(* CoDeSys 2.3.9.47 project: wtp_sfc_6_1_2016.pro *)
(* Libraries: TcSystem.lib 21.1.15 10:22:54, TcBase.lib 14.5.09 12:14:08, TcUtilities.lib 6.1.15 16:45:04, TcBABasic.lib 22.7.15 15:46:14, STANDARD.LIB 5.6.98 12:03:02 *)

(* Task configuration *)
TASK Standard (PRIORITY := 0, INTERVAL := T#500ms);
	MAIN
END_TASK

(* POU MAIN, ST *)
PROGRAM MAIN
VAR
(*EQUALISATION TRANSFER*)

	InletEqPumpOp1 :  INLET_EQ_PUMP;

	LSL101A: BOOL;
	LSS101A: BOOL;
	LSH101A: BOOL;
	LSD101A: BOOL;
	LSHH105A: BOOL;
	LSH103A: BOOL;
	LSS103A: BOOL;

	InletEqPumpOp2 :  INLET_EQ_PUMP;

	LSL101B: BOOL;
	LSS101B: BOOL;
	LSH101B: BOOL;
	LSD101B: BOOL;
	LSHH105B: BOOL;
	LSH103B: BOOL;
	LSS103B: BOOL;


	InletMixerOp1 : INLET_MIXER;
	LSL100A : BOOL;
	LSHL100A : BOOL;

	InletMixerOp2 : INLET_MIXER;
	LSL100B : BOOL;
	LSHL100B : BOOL;


(*SBR TRANSFER*)
	SBRTrans_OP1_InletSBRTrans : INLET_EQ_PUMP;
	SBRTrans_OP2_InletSBRTrans : INLET_EQ_PUMP;

	test : DEVICES_DOUBLE_DUTY;
	WaterPressureSensor: REAL;

(*Reuse Water Syatem*)
	Reuse_Water_System : REUSE_WATER_SYS;

(*Screen House*)
	ScreenOperation1 : SCREENING_OPERATION;


END_VAR
(*EQUALISATION TRANSFER*)
InletEqPumpOp1(
	sigEQFloatSensorLO:= LSL101A,
	sigEQFLoatSensorOP:= LSS101A,
	sigEQFloatSensorHi:= LSH101A,
	sigEQFLoatSensorDry:= LSD101A,
	sigStreamLineOverFLow:=LSHH105A ,
	sigSBRFloatSensorHi:= LSH103A,
	sigSBRFloatSensorOP:=LSS103A );

InletEqPumpOp2(
	sigEQFloatSensorLO:= LSL101B,
	sigEQFLoatSensorOP:= LSS101B,
	sigEQFloatSensorHi:= LSH101B,
	sigEQFLoatSensorDry:= LSD101B,
	sigStreamLineOverFLow:=LSHH105B ,
	sigSBRFloatSensorHi:= LSH103B,
	sigSBRFloatSensorOP:=LSS103B );

InletMixerOp1(sigMixerFloatSensorLO:=LSL100A , sigMixerFloatSensorHI:=LSHL100A );

InletMixerOp2(sigMixerFloatSensorLO:=LSL100B , sigMixerFloatSensorHI:=LSHL100B );



(*Reuse Water Syatem*)
	Reuse_Water_System();



(*Screen House*)
ScreenOperation1();
END_PROGRAM

(* POU INLET_EQ_PUMP, SFC *)
FUNCTION_BLOCK  INLET_EQ_PUMP
VAR

	Reset : BOOL;
	CriticalAlarm_FloatSensorHi : BOOL;
	CriticalAlarm_FloatSensorDRY : BOOL;
	Warning_FloatSensorDry : BOOL;


	Pump : DEVICES_DUTY_STANDBY;

	Act_Reset : BOOL;
	Act_Start : BOOL;
	Act_Stop : BOOL;

	FB_Contacts_1: FB_Contacts;
	FB_Contacts_2:FB_Contacts;
	FB_Contacts_3:FB_Contacts;
	FB_Contacts_4:FB_Contacts;
	FB_Contacts_5:FB_Contacts;
	FB_Contacts_6:FB_Contacts;
	FB_Contacts_7:FB_Contacts;


	EQFloatSensorLO : BOOL;
	EQFLoatSensorOP : BOOL;
	EQFloatSensorHi : BOOL;
	EQFLoatSensorDry : BOOL;
	StreamLineOverFLow : BOOL;
	SBRFloatSensorHi : BOOL;
	SBRFloatSensorOP : BOOL;
END_VAR
VAR_IN_OUT
	sigEQFloatSensorLO : BOOL;
	sigEQFLoatSensorOP : BOOL;
	sigEQFloatSensorHi : BOOL;
	sigEQFLoatSensorDry : BOOL;
	sigStreamLineOverFLow : BOOL;
	sigSBRFloatSensorHi : BOOL;
	sigSBRFloatSensorOP : BOOL;
END_VAR
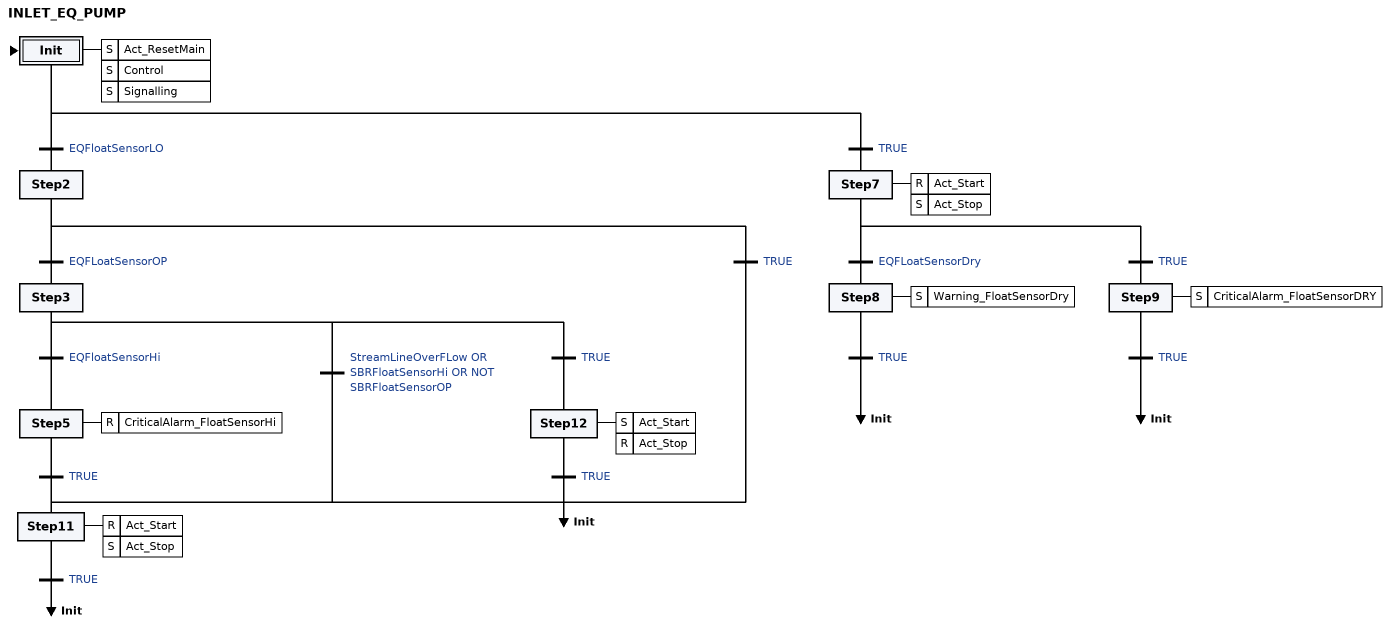
INITIAL_STEP Init:
	Act_ResetMain(S);
	Control(S);
	Signalling(S);
END_STEP
TRANSITION FROM Init TO Step2 := EQFloatSensorLO;
END_TRANSITION
TRANSITION FROM Init TO Step7 := TRUE;
END_TRANSITION
STEP Step2:
END_STEP
TRANSITION FROM Step2 TO Step3 := EQFLoatSensorOP;
END_TRANSITION
TRANSITION FROM Step2 TO Step11 := TRUE;
END_TRANSITION
STEP Step3:
END_STEP
TRANSITION FROM Step3 TO Step5 := EQFloatSensorHi;
END_TRANSITION
TRANSITION FROM Step3 TO Step11 := StreamLineOverFLow OR SBRFloatSensorHi OR NOT SBRFloatSensorOP;
END_TRANSITION
TRANSITION FROM Step3 TO Step12 := TRUE;
END_TRANSITION
STEP Step5:
	CriticalAlarm_FloatSensorHi(R);
END_STEP
TRANSITION FROM Step5 TO Step11 := TRUE;
END_TRANSITION
STEP Step11:
	Act_Start(R);
	Act_Stop(S);
END_STEP
TRANSITION FROM Step11 TO Init := TRUE;
END_TRANSITION
STEP Step12:
	Act_Start(S);
	Act_Stop(R);
END_STEP
TRANSITION FROM Step12 TO Init := TRUE;
END_TRANSITION
STEP Step7:
	Act_Start(R);
	Act_Stop(S);
END_STEP
TRANSITION FROM Step7 TO Step8 := EQFLoatSensorDry;
END_TRANSITION
TRANSITION FROM Step7 TO Step9 := TRUE;
END_TRANSITION
STEP Step8:
	Warning_FloatSensorDry(S);
END_STEP
TRANSITION FROM Step8 TO Init := TRUE;
END_TRANSITION
STEP Step9:
	CriticalAlarm_FloatSensorDRY(S);
END_STEP
TRANSITION FROM Step9 TO Init := TRUE;
END_TRANSITION
END_FUNCTION_BLOCK
ACTION Act_ResetMain:
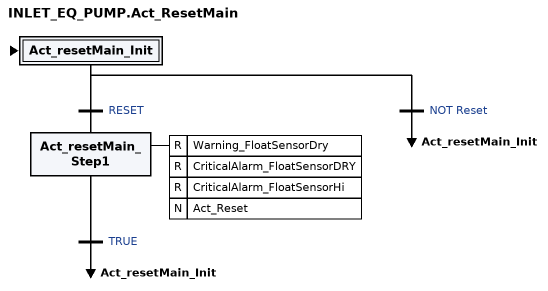
INITIAL_STEP Act_resetMain_Init:
END_STEP
TRANSITION FROM Act_resetMain_Init TO Act_resetMain_Step1 := RESET;
END_TRANSITION
TRANSITION FROM Act_resetMain_Init TO Act_resetMain_Init := NOT Reset;
END_TRANSITION
STEP Act_resetMain_Step1:
	Warning_FloatSensorDry(R);
	CriticalAlarm_FloatSensorDRY(R);
	CriticalAlarm_FloatSensorHi(R);
	Act_Reset(N);
END_STEP
TRANSITION FROM Act_resetMain_Step1 TO Act_resetMain_Init := TRUE;
END_TRANSITION
END_ACTION
ACTION Control:
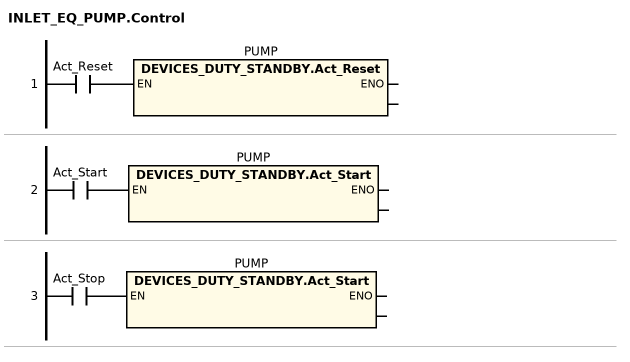
_LD_ (* Ladder Diagram *)
NETWORK 1
	[Act_Reset]
		EN --- PUMP:DEVICES_DUTY_STANDBY.Act_Reset()
NETWORK 2
	[Act_Start]
		EN --- PUMP:DEVICES_DUTY_STANDBY.Act_Start()
NETWORK 3
	[Act_Stop]
		EN --- PUMP:DEVICES_DUTY_STANDBY.Act_Start()
_END_LD_
(* the same logic as Structured Text *)
(* Network 1 *)
IF Act_Reset THEN
	PUMP();
END_IF;
(* Network 2 *)
IF Act_Start THEN
	PUMP();
END_IF;
(* Network 3 *)
IF Act_Stop THEN
	PUMP();
END_IF;
END_ACTION
ACTION Signalling:
FB_Contacts_1(IN:=sigEQFloatSensorLO ,Q=> EQFloatSensorLO);
FB_Contacts_2(IN:=sigEQFLoatSensorOP ,Q=> EQFLoatSensorOP);
FB_Contacts_3(IN:=sigEQFloatSensorHi ,Q=> EQFloatSensorHi);
FB_Contacts_4(IN:=sigEQFLoatSensorDry ,Q=> EQFLoatSensorDry);
FB_Contacts_5(IN:=sigStreamLineOverFLow ,Q=> StreamLineOverFLow);
FB_Contacts_6(IN:=sigSBRFloatSensorHi ,Q=> SBRFloatSensorHi);
FB_Contacts_7(IN:=sigSBRFloatSensorOP ,Q=> SBRFloatSensorOP);
END_ACTION

(* POU DEVICES_DUTY_STANDBY, SFC *)
FUNCTION_BLOCK DEVICES_DUTY_STANDBY
VAR


	Duty_RemoteMode AT%I*: BOOL;
	Duty_CommandStart AT%I*: BOOL;
	Duty_Overload AT%I*: BOOL;
	Duty_Incomplete AT%I*: BOOL;
	Duty_StartStatus AT%I*: BOOL;


	Done_StartStandby: BOOL;
	Done_Start: BOOL;
	Done_Stop: BOOL;


	Standby_CommandStart AT%I*: BOOL;
	Standby_RemoteMode AT%I*: BOOL;
	Standby_Overload AT%I*: BOOL;
	Standby_Incomplete AT%I*: BOOL;
	Standby_StartStatus AT%I*: BOOL;


	Warning_DutyFailed: BOOL;
	Warning_StandbyFailed: BOOL;
	CriticalAlarm_StandbyCannotStop : BOOL;
	CriticalAlarm_DutyCannotStop : BOOL;
	CriticalAlarm_DutyStandbyFailedToStart: BOOL;

END_VAR
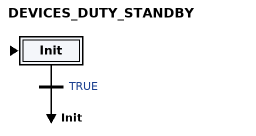
INITIAL_STEP Init:
END_STEP
TRANSITION FROM Init TO Init := TRUE;
END_TRANSITION
END_FUNCTION_BLOCK
ACTION Act_Reset:
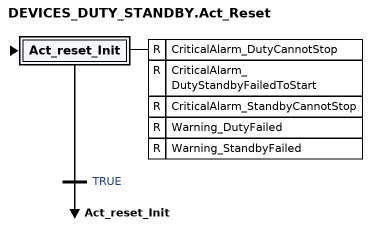
INITIAL_STEP Act_reset_Init:
	CriticalAlarm_DutyCannotStop(R);
	CriticalAlarm_DutyStandbyFailedToStart(R);
	CriticalAlarm_StandbyCannotStop(R);
	Warning_DutyFailed(R);
	Warning_StandbyFailed(R);
END_STEP
TRANSITION FROM Act_reset_Init TO Act_reset_Init := TRUE;
END_TRANSITION
END_ACTION
ACTION Act_Start:
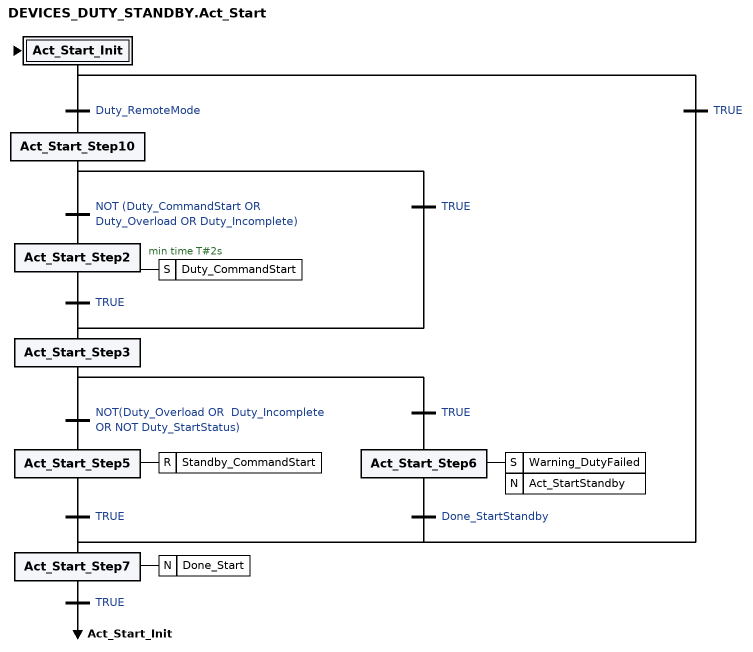
INITIAL_STEP Act_Start_Init:
END_STEP
TRANSITION FROM Act_Start_Init TO Act_Start_Step10 := Duty_RemoteMode;
END_TRANSITION
TRANSITION FROM Act_Start_Init TO Act_Start_Step7 := TRUE;
END_TRANSITION
STEP Act_Start_Step10:
END_STEP
TRANSITION FROM Act_Start_Step10 TO Act_Start_Step2 := NOT (Duty_CommandStart OR Duty_Overload OR Duty_Incomplete);
END_TRANSITION
TRANSITION FROM Act_Start_Step10 TO Act_Start_Step3 := TRUE;
END_TRANSITION
STEP Act_Start_Step2: (* min time T#2s *)
	Duty_CommandStart(S);
END_STEP
TRANSITION FROM Act_Start_Step2 TO Act_Start_Step3 := TRUE;
END_TRANSITION
STEP Act_Start_Step3:
END_STEP
TRANSITION FROM Act_Start_Step3 TO Act_Start_Step5 := NOT(Duty_Overload OR  Duty_Incomplete OR NOT Duty_StartStatus);
END_TRANSITION
TRANSITION FROM Act_Start_Step3 TO Act_Start_Step6 := TRUE;
END_TRANSITION
STEP Act_Start_Step5:
	Standby_CommandStart(R);
END_STEP
TRANSITION FROM Act_Start_Step5 TO Act_Start_Step7 := TRUE;
END_TRANSITION
STEP Act_Start_Step6:
	Warning_DutyFailed(S);
	Act_StartStandby(N);
END_STEP
TRANSITION FROM Act_Start_Step6 TO Act_Start_Step7 := Done_StartStandby;
END_TRANSITION
STEP Act_Start_Step7:
	Done_Start(N);
END_STEP
TRANSITION FROM Act_Start_Step7 TO Act_Start_Init := TRUE;
END_TRANSITION
END_ACTION
ACTION Act_StartStandby:
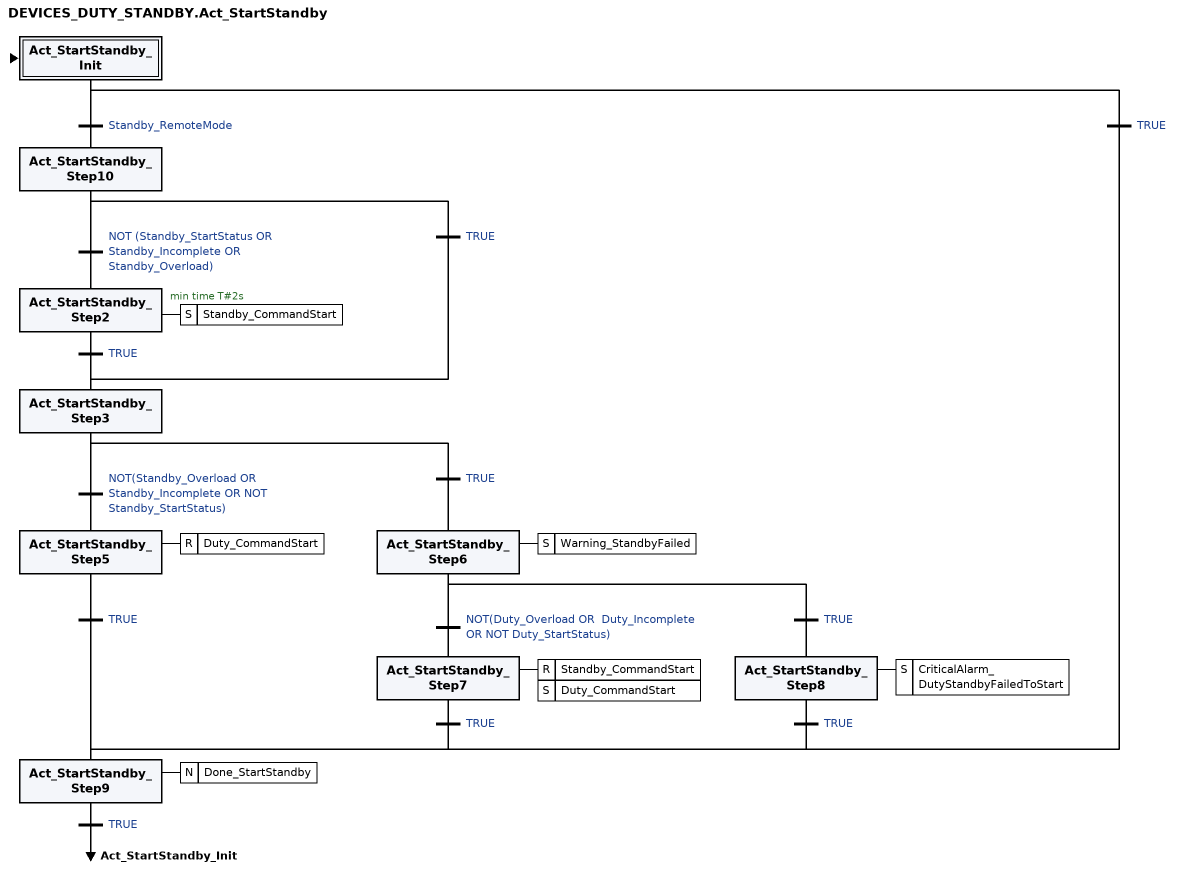
INITIAL_STEP Act_StartStandby_Init:
END_STEP
TRANSITION FROM Act_StartStandby_Init TO Act_StartStandby_Step10 := Standby_RemoteMode;
END_TRANSITION
TRANSITION FROM Act_StartStandby_Init TO Act_StartStandby_Step9 := TRUE;
END_TRANSITION
STEP Act_StartStandby_Step10:
END_STEP
TRANSITION FROM Act_StartStandby_Step10 TO Act_StartStandby_Step2 := NOT (Standby_StartStatus OR Standby_Incomplete OR Standby_Overload);
END_TRANSITION
TRANSITION FROM Act_StartStandby_Step10 TO Act_StartStandby_Step3 := TRUE;
END_TRANSITION
STEP Act_StartStandby_Step2: (* min time T#2s *)
	Standby_CommandStart(S);
END_STEP
TRANSITION FROM Act_StartStandby_Step2 TO Act_StartStandby_Step3 := TRUE;
END_TRANSITION
STEP Act_StartStandby_Step3:
END_STEP
TRANSITION FROM Act_StartStandby_Step3 TO Act_StartStandby_Step5 := NOT(Standby_Overload OR  Standby_Incomplete OR NOT Standby_StartStatus);
END_TRANSITION
TRANSITION FROM Act_StartStandby_Step3 TO Act_StartStandby_Step6 := TRUE;
END_TRANSITION
STEP Act_StartStandby_Step5:
	Duty_CommandStart(R);
END_STEP
TRANSITION FROM Act_StartStandby_Step5 TO Act_StartStandby_Step9 := TRUE;
END_TRANSITION
STEP Act_StartStandby_Step6:
	Warning_StandbyFailed(S);
END_STEP
TRANSITION FROM Act_StartStandby_Step6 TO Act_StartStandby_Step7 := NOT(Duty_Overload OR  Duty_Incomplete OR NOT Duty_StartStatus);
END_TRANSITION
TRANSITION FROM Act_StartStandby_Step6 TO Act_StartStandby_Step8 := TRUE;
END_TRANSITION
STEP Act_StartStandby_Step7:
	Standby_CommandStart(R);
	Duty_CommandStart(S);
END_STEP
TRANSITION FROM Act_StartStandby_Step7 TO Act_StartStandby_Step9 := TRUE;
END_TRANSITION
STEP Act_StartStandby_Step8:
	CriticalAlarm_DutyStandbyFailedToStart (S);
END_STEP
TRANSITION FROM Act_StartStandby_Step8 TO Act_StartStandby_Step9 := TRUE;
END_TRANSITION
STEP Act_StartStandby_Step9:
	Done_StartStandby(N);
END_STEP
TRANSITION FROM Act_StartStandby_Step9 TO Act_StartStandby_Init := TRUE;
END_TRANSITION
END_ACTION
ACTION Act_Stop:
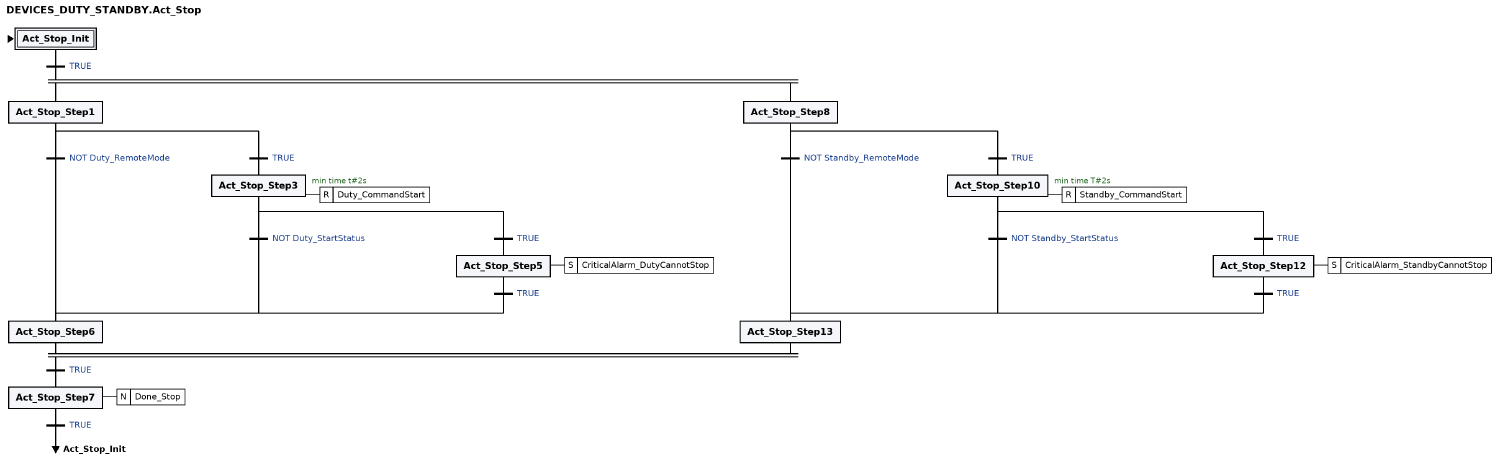
INITIAL_STEP Act_Stop_Init:
END_STEP
TRANSITION FROM Act_Stop_Init TO (Act_Stop_Step1, Act_Stop_Step8) := TRUE;
END_TRANSITION
STEP Act_Stop_Step1:
END_STEP
TRANSITION FROM Act_Stop_Step1 TO Act_Stop_Step6 := NOT Duty_RemoteMode;
END_TRANSITION
TRANSITION FROM Act_Stop_Step1 TO Act_Stop_Step3 := TRUE;
END_TRANSITION
STEP Act_Stop_Step3: (* min time t#2s *)
	Duty_CommandStart(R);
END_STEP
TRANSITION FROM Act_Stop_Step3 TO Act_Stop_Step6 := NOT Duty_StartStatus;
END_TRANSITION
TRANSITION FROM Act_Stop_Step3 TO Act_Stop_Step5 := TRUE;
END_TRANSITION
STEP Act_Stop_Step5:
	CriticalAlarm_DutyCannotStop(S);
END_STEP
TRANSITION FROM Act_Stop_Step5 TO Act_Stop_Step6 := TRUE;
END_TRANSITION
STEP Act_Stop_Step6:
END_STEP
STEP Act_Stop_Step8:
END_STEP
TRANSITION FROM Act_Stop_Step8 TO Act_Stop_Step13 := NOT Standby_RemoteMode;
END_TRANSITION
TRANSITION FROM Act_Stop_Step8 TO Act_Stop_Step10 := TRUE;
END_TRANSITION
STEP Act_Stop_Step10: (* min time T#2s *)
	Standby_CommandStart(R);
END_STEP
TRANSITION FROM Act_Stop_Step10 TO Act_Stop_Step13 := NOT Standby_StartStatus;
END_TRANSITION
TRANSITION FROM Act_Stop_Step10 TO Act_Stop_Step12 := TRUE;
END_TRANSITION
STEP Act_Stop_Step12:
	CriticalAlarm_StandbyCannotStop(S);
END_STEP
TRANSITION FROM Act_Stop_Step12 TO Act_Stop_Step13 := TRUE;
END_TRANSITION
STEP Act_Stop_Step13:
END_STEP
TRANSITION FROM (Act_Stop_Step6, Act_Stop_Step13) TO Act_Stop_Step7 := TRUE;
END_TRANSITION
STEP Act_Stop_Step7:
	Done_Stop(N);
END_STEP
TRANSITION FROM Act_Stop_Step7 TO Act_Stop_Init := TRUE;
END_TRANSITION
END_ACTION

(* POU FB_Contacts, ST *)
FUNCTION_BLOCK FB_Contacts
VAR_INPUT
	IN: BOOL;
END_VAR
VAR_OUTPUT
	Q : BOOL;
END_VAR
VAR
	FBThresholdSwitch: FB_ThresholdSwitch;
END_VAR
IF IN THEN
FBThresholdSwitch.fSignal := 1;
ELSE
FBThresholdSwitch.fSignal := 0;
END_IF

FBThresholdSwitch(
	fLowerLimit:=0,
	fUpperLimit:=1,
	tLowerLimitDelay:=T#5s,
	tUpperLimitDelay:=T#5s ,
	bSwitchingSignal=>Q ,
	bCrossLowerLimit=> , 
	bCrossUpperLimit=> );
END_FUNCTION_BLOCK

(* POU INLET_MIXER, SFC *)
FUNCTION_BLOCK INLET_MIXER
VAR

	MixerFloatSensorLO: BOOL;
	MixerFloatSensorHI : BOOL;
	Mixer : DEVICES_DUTY_STANDBY;

	FB_Contacts_1: FB_Contacts;
	FB_Contacts_2: FB_Contacts;

	Reset : BOOL;
	Act_Reset : BOOL;
	Act_Start : BOOL;
	Act_Stop : BOOL;
END_VAR

VAR_IN_OUT
	sigMixerFloatSensorLO: BOOL;
	sigMixerFloatSensorHI : BOOL;
END_VAR
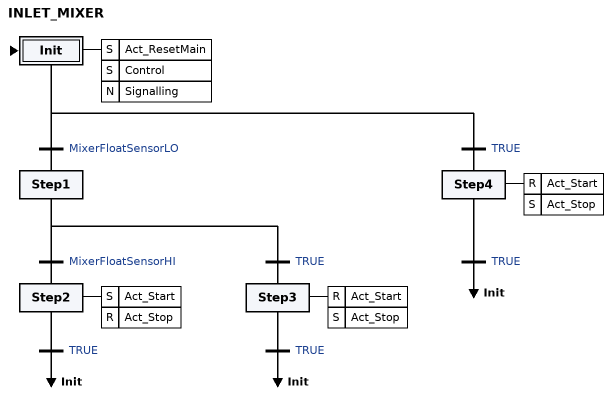
INITIAL_STEP Init:
	Act_ResetMain(S);
	Control(S);
	Signalling(N);
END_STEP
TRANSITION FROM Init TO Step1 := MixerFloatSensorLO;
END_TRANSITION
TRANSITION FROM Init TO Step4 := TRUE;
END_TRANSITION
STEP Step1:
END_STEP
TRANSITION FROM Step1 TO Step2 := MixerFloatSensorHI;
END_TRANSITION
TRANSITION FROM Step1 TO Step3 := TRUE;
END_TRANSITION
STEP Step2:
	Act_Start(S);
	Act_Stop(R);
END_STEP
TRANSITION FROM Step2 TO Init := TRUE;
END_TRANSITION
STEP Step3:
	Act_Start(R);
	Act_Stop(S);
END_STEP
TRANSITION FROM Step3 TO Init := TRUE;
END_TRANSITION
STEP Step4:
	Act_Start(R);
	Act_Stop(S);
END_STEP
TRANSITION FROM Step4 TO Init := TRUE;
END_TRANSITION
END_FUNCTION_BLOCK
ACTION Act_ResetMain:
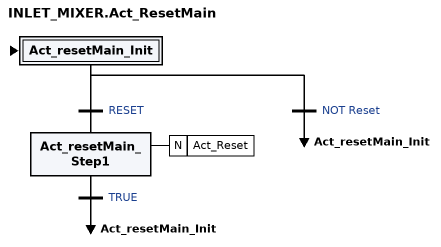
INITIAL_STEP Act_resetMain_Init:
END_STEP
TRANSITION FROM Act_resetMain_Init TO Act_resetMain_Step1 := RESET;
END_TRANSITION
TRANSITION FROM Act_resetMain_Init TO Act_resetMain_Init := NOT Reset;
END_TRANSITION
STEP Act_resetMain_Step1:
	Act_Reset(N);
END_STEP
TRANSITION FROM Act_resetMain_Step1 TO Act_resetMain_Init := TRUE;
END_TRANSITION
END_ACTION
ACTION Control:
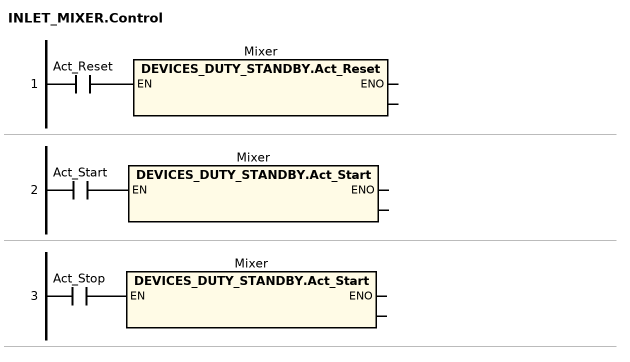
_LD_ (* Ladder Diagram *)
NETWORK 1
	[Act_Reset]
		EN --- Mixer:DEVICES_DUTY_STANDBY.Act_Reset()
NETWORK 2
	[Act_Start]
		EN --- Mixer:DEVICES_DUTY_STANDBY.Act_Start()
NETWORK 3
	[Act_Stop]
		EN --- Mixer:DEVICES_DUTY_STANDBY.Act_Start()
_END_LD_
(* the same logic as Structured Text *)
(* Network 1 *)
IF Act_Reset THEN
	Mixer();
END_IF;
(* Network 2 *)
IF Act_Start THEN
	Mixer();
END_IF;
(* Network 3 *)
IF Act_Stop THEN
	Mixer();
END_IF;
END_ACTION
ACTION Signalling:
FB_Contacts_1(IN:=sigMixerFloatSensorLO ,Q=> MixerFloatSensorLO);
FB_Contacts_2(IN:=sigMixerFloatSensorHI ,Q=> MixerFloatSensorHI);
END_ACTION

(* POU DEVICES_DOUBLE_DUTY, SFC *)
FUNCTION_BLOCK DEVICES_DOUBLE_DUTY
VAR

	Duty_RemoteMode AT%I*: BOOL;
	Duty_CommandStart AT%I*: BOOL;
	Duty_Overload AT%I*: BOOL;
	Duty_Incomplete AT%I*: BOOL;
	Duty_StartStatus AT%I*: BOOL;


	Done_StartStandby: BOOL;
	Done_Start: BOOL;
	Done_Stop: BOOL;


	Duty2_CommandStart AT%I*: BOOL;
	Duty2_RemoteMode AT%I*: BOOL;
	Duty2_Overload AT%I*: BOOL;
	Duty2_Incomplete AT%I*: BOOL;
	Duty2_StartStatus AT%I*: BOOL;

	Warning_DutyFailed: BOOL;
	Warning_Duty2Failed: BOOL;
	CriticalAlarm_Duty2CannotStop : BOOL;
	CriticalAlarm_DutyCannotStop : BOOL;

END_VAR
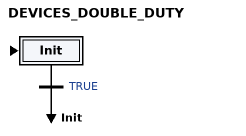
INITIAL_STEP Init:
END_STEP
TRANSITION FROM Init TO Init := TRUE;
END_TRANSITION
END_FUNCTION_BLOCK
ACTION Act_Reset:
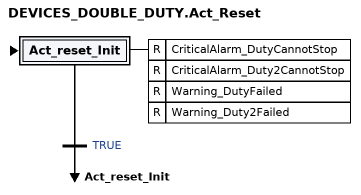
INITIAL_STEP Act_reset_Init:
	CriticalAlarm_DutyCannotStop(R);
	CriticalAlarm_Duty2CannotStop(R);
	Warning_DutyFailed(R);
	Warning_Duty2Failed(R);
END_STEP
TRANSITION FROM Act_reset_Init TO Act_reset_Init := TRUE;
END_TRANSITION
END_ACTION
ACTION Act_Start:
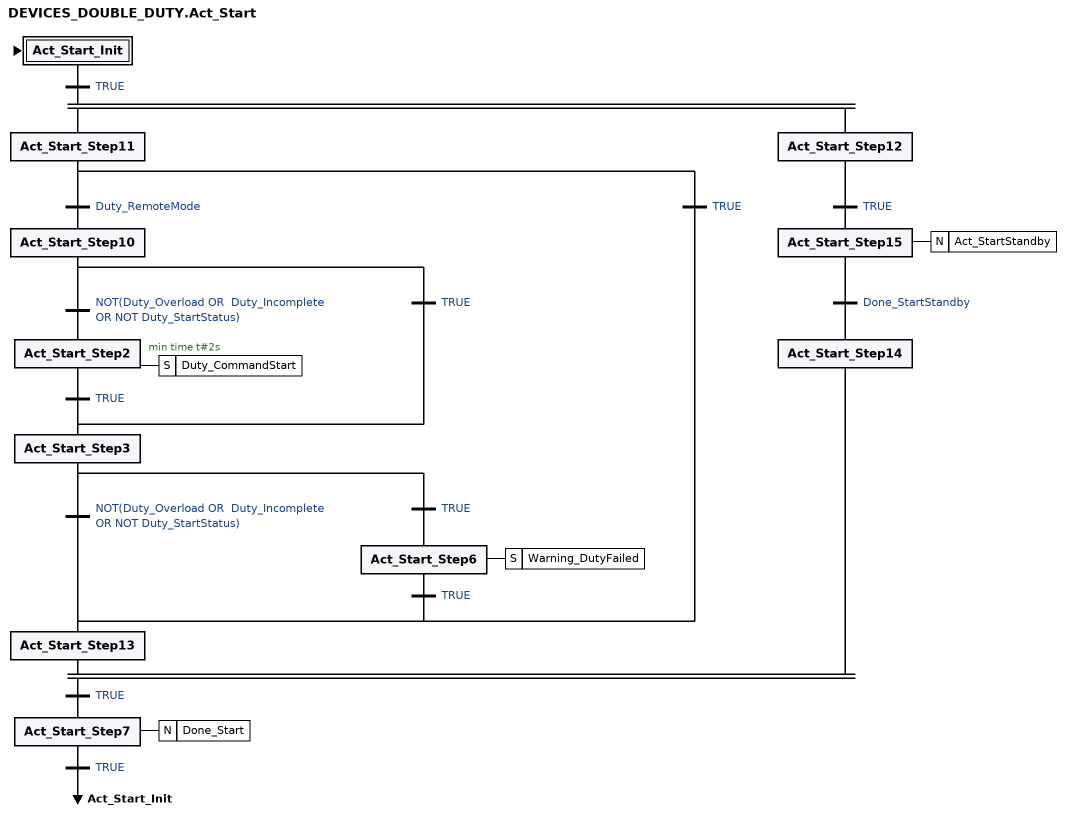
INITIAL_STEP Act_Start_Init:
END_STEP
TRANSITION FROM Act_Start_Init TO (Act_Start_Step11, Act_Start_Step12) := TRUE;
END_TRANSITION
STEP Act_Start_Step11:
END_STEP
TRANSITION FROM Act_Start_Step11 TO Act_Start_Step10 := Duty_RemoteMode;
END_TRANSITION
TRANSITION FROM Act_Start_Step11 TO Act_Start_Step13 := TRUE;
END_TRANSITION
STEP Act_Start_Step10:
END_STEP
TRANSITION FROM Act_Start_Step10 TO Act_Start_Step2 := NOT(Duty_Overload OR  Duty_Incomplete OR NOT Duty_StartStatus);
END_TRANSITION
TRANSITION FROM Act_Start_Step10 TO Act_Start_Step3 := TRUE;
END_TRANSITION
STEP Act_Start_Step2: (* min time t#2s *)
	Duty_CommandStart(S);
END_STEP
TRANSITION FROM Act_Start_Step2 TO Act_Start_Step3 := TRUE;
END_TRANSITION
STEP Act_Start_Step3:
END_STEP
TRANSITION FROM Act_Start_Step3 TO Act_Start_Step13 := NOT(Duty_Overload OR  Duty_Incomplete OR NOT Duty_StartStatus);
END_TRANSITION
TRANSITION FROM Act_Start_Step3 TO Act_Start_Step6 := TRUE;
END_TRANSITION
STEP Act_Start_Step6:
	Warning_DutyFailed(S);
END_STEP
TRANSITION FROM Act_Start_Step6 TO Act_Start_Step13 := TRUE;
END_TRANSITION
STEP Act_Start_Step13:
END_STEP
STEP Act_Start_Step12:
END_STEP
TRANSITION FROM Act_Start_Step12 TO Act_Start_Step15 := TRUE;
END_TRANSITION
STEP Act_Start_Step15:
	Act_StartStandby(N);
END_STEP
TRANSITION FROM Act_Start_Step15 TO Act_Start_Step14 := Done_StartStandby;
END_TRANSITION
STEP Act_Start_Step14:
END_STEP
TRANSITION FROM (Act_Start_Step13, Act_Start_Step14) TO Act_Start_Step7 := TRUE;
END_TRANSITION
STEP Act_Start_Step7:
	Done_Start(N);
END_STEP
TRANSITION FROM Act_Start_Step7 TO Act_Start_Init := TRUE;
END_TRANSITION
END_ACTION
ACTION Act_StartStandby:
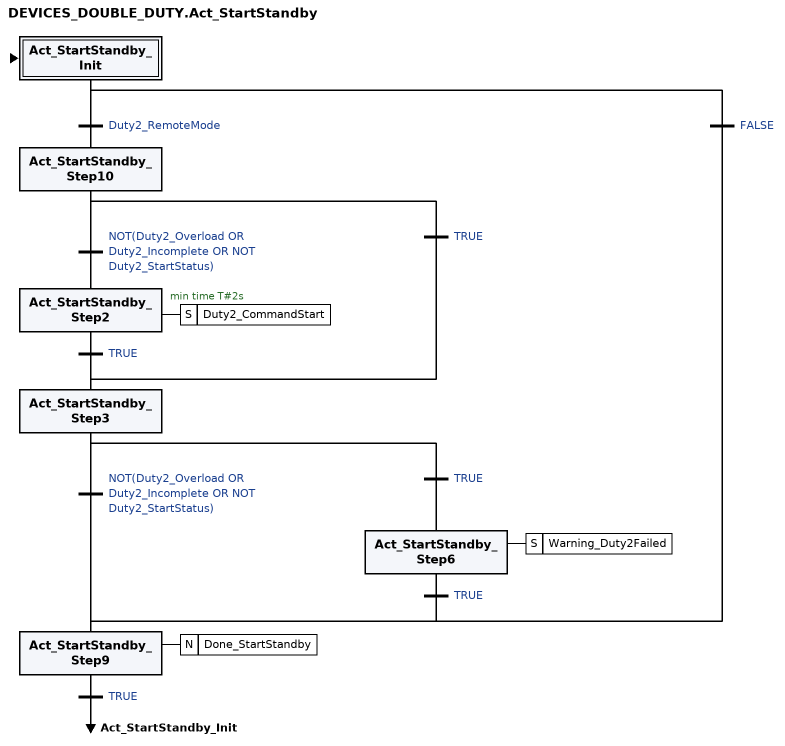
INITIAL_STEP Act_StartStandby_Init:
END_STEP
TRANSITION FROM Act_StartStandby_Init TO Act_StartStandby_Step10 := Duty2_RemoteMode;
END_TRANSITION
TRANSITION FROM Act_StartStandby_Init TO Act_StartStandby_Step9 := FALSE;
END_TRANSITION
STEP Act_StartStandby_Step10:
END_STEP
TRANSITION FROM Act_StartStandby_Step10 TO Act_StartStandby_Step2 := NOT(Duty2_Overload OR  Duty2_Incomplete OR NOT Duty2_StartStatus);
END_TRANSITION
TRANSITION FROM Act_StartStandby_Step10 TO Act_StartStandby_Step3 := TRUE;
END_TRANSITION
STEP Act_StartStandby_Step2: (* min time T#2s *)
	Duty2_CommandStart(S);
END_STEP
TRANSITION FROM Act_StartStandby_Step2 TO Act_StartStandby_Step3 := TRUE;
END_TRANSITION
STEP Act_StartStandby_Step3:
END_STEP
TRANSITION FROM Act_StartStandby_Step3 TO Act_StartStandby_Step9 := NOT(Duty2_Overload OR  Duty2_Incomplete OR NOT Duty2_StartStatus);
END_TRANSITION
TRANSITION FROM Act_StartStandby_Step3 TO Act_StartStandby_Step6 := TRUE;
END_TRANSITION
STEP Act_StartStandby_Step6:
	Warning_Duty2Failed(S);
END_STEP
TRANSITION FROM Act_StartStandby_Step6 TO Act_StartStandby_Step9 := TRUE;
END_TRANSITION
STEP Act_StartStandby_Step9:
	Done_StartStandby(N);
END_STEP
TRANSITION FROM Act_StartStandby_Step9 TO Act_StartStandby_Init := TRUE;
END_TRANSITION
END_ACTION
ACTION Act_Stop:
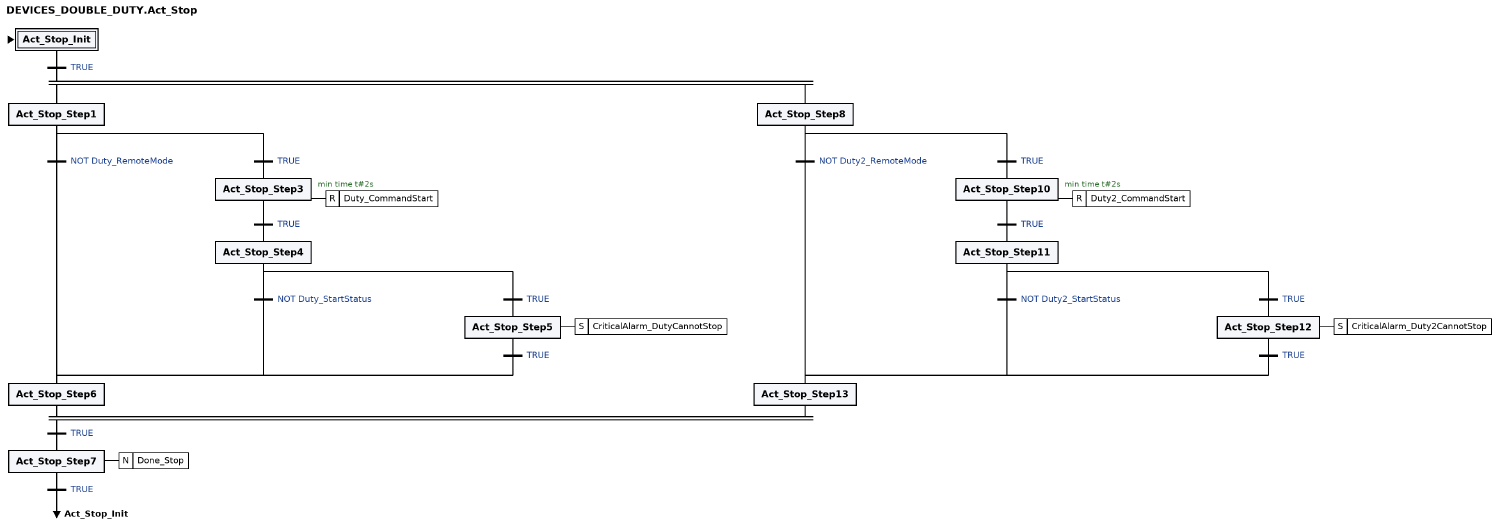
INITIAL_STEP Act_Stop_Init:
END_STEP
TRANSITION FROM Act_Stop_Init TO (Act_Stop_Step1, Act_Stop_Step8) := TRUE;
END_TRANSITION
STEP Act_Stop_Step1:
END_STEP
TRANSITION FROM Act_Stop_Step1 TO Act_Stop_Step6 := NOT Duty_RemoteMode;
END_TRANSITION
TRANSITION FROM Act_Stop_Step1 TO Act_Stop_Step3 := TRUE;
END_TRANSITION
STEP Act_Stop_Step3: (* min time t#2s *)
	Duty_CommandStart(R);
END_STEP
TRANSITION FROM Act_Stop_Step3 TO Act_Stop_Step4 := TRUE;
END_TRANSITION
STEP Act_Stop_Step4:
END_STEP
TRANSITION FROM Act_Stop_Step4 TO Act_Stop_Step6 := NOT Duty_StartStatus;
END_TRANSITION
TRANSITION FROM Act_Stop_Step4 TO Act_Stop_Step5 := TRUE;
END_TRANSITION
STEP Act_Stop_Step5:
	CriticalAlarm_DutyCannotStop(S);
END_STEP
TRANSITION FROM Act_Stop_Step5 TO Act_Stop_Step6 := TRUE;
END_TRANSITION
STEP Act_Stop_Step6:
END_STEP
STEP Act_Stop_Step8:
END_STEP
TRANSITION FROM Act_Stop_Step8 TO Act_Stop_Step13 := NOT Duty2_RemoteMode;
END_TRANSITION
TRANSITION FROM Act_Stop_Step8 TO Act_Stop_Step10 := TRUE;
END_TRANSITION
STEP Act_Stop_Step10: (* min time t#2s *)
	Duty2_CommandStart(R);
END_STEP
TRANSITION FROM Act_Stop_Step10 TO Act_Stop_Step11 := TRUE;
END_TRANSITION
STEP Act_Stop_Step11:
END_STEP
TRANSITION FROM Act_Stop_Step11 TO Act_Stop_Step13 := NOT Duty2_StartStatus;
END_TRANSITION
TRANSITION FROM Act_Stop_Step11 TO Act_Stop_Step12 := TRUE;
END_TRANSITION
STEP Act_Stop_Step12:
	CriticalAlarm_Duty2CannotStop(S);
END_STEP
TRANSITION FROM Act_Stop_Step12 TO Act_Stop_Step13 := TRUE;
END_TRANSITION
STEP Act_Stop_Step13:
END_STEP
TRANSITION FROM (Act_Stop_Step6, Act_Stop_Step13) TO Act_Stop_Step7 := TRUE;
END_TRANSITION
STEP Act_Stop_Step7:
	Done_Stop(N);
END_STEP
TRANSITION FROM Act_Stop_Step7 TO Act_Stop_Init := TRUE;
END_TRANSITION
END_ACTION

(* POU REUSE_WATER_SYS, SFC *)
FUNCTION_BLOCK REUSE_WATER_SYS
VAR_INPUT
END_VAR
VAR_OUTPUT
END_VAR
VAR
	VacumPump_AB : DEVICES_DUTY_STANDBY;
	LeadPump_AB : DEVICES_DOUBLE_DUTY;
	LeadPump_CD: DEVICES_DOUBLE_DUTY;
	JockeyPump_AB : DEVICES_DUTY_STANDBY;
	LSL308A AT%I*: BOOL;
	LSH308B AT%I*: BOOL;
	LSL308B AT%I*: BOOL;
	LSH308A AT%I*: BOOL;
	Done_Active: BOOL;
	XV101 AT%Q* : BOOL;
	XV102 AT%Q*: BOOL;
	Done_Vacum_Priming: BOOL;
	Done_On_Pump_Seq: BOOL;
	LSH406 AT%I*: BOOL;
	FSL101 AT%I*: BOOL;
	LSH405 AT%I*: BOOL;
	WaterPressureSensor: LREAL;
	Timer1: TON;
	done_TimerWaterPressure: BOOL;
	Reset_TimerWaterPressure: BOOL;
	WarningAlarm_HighPressure : BOOL;
	Done_stop: BOOL;
	RESET: BOOL;
	Act_JockeyPump_AB_Reset: BOOL;
	Act_JockeyPump_AB_Start: BOOL;
	Act_JockeyPump_AB_Stop: BOOL;
	Act_LeadPump_AB_Reset: BOOL;
	Act_LeadPump_AB_Start: BOOL;
	Act_LeadPump_AB_Stop: BOOL;
	Act_LeadPump_CD_Reset: BOOL;
	Act_LeadPump_CD_Start: BOOL;
	Act_LeadPump_CD_Stop: BOOL;
	Set_TimerWaterPressure: BOOL;
	Error_DryRun: BOOL;
END_VAR
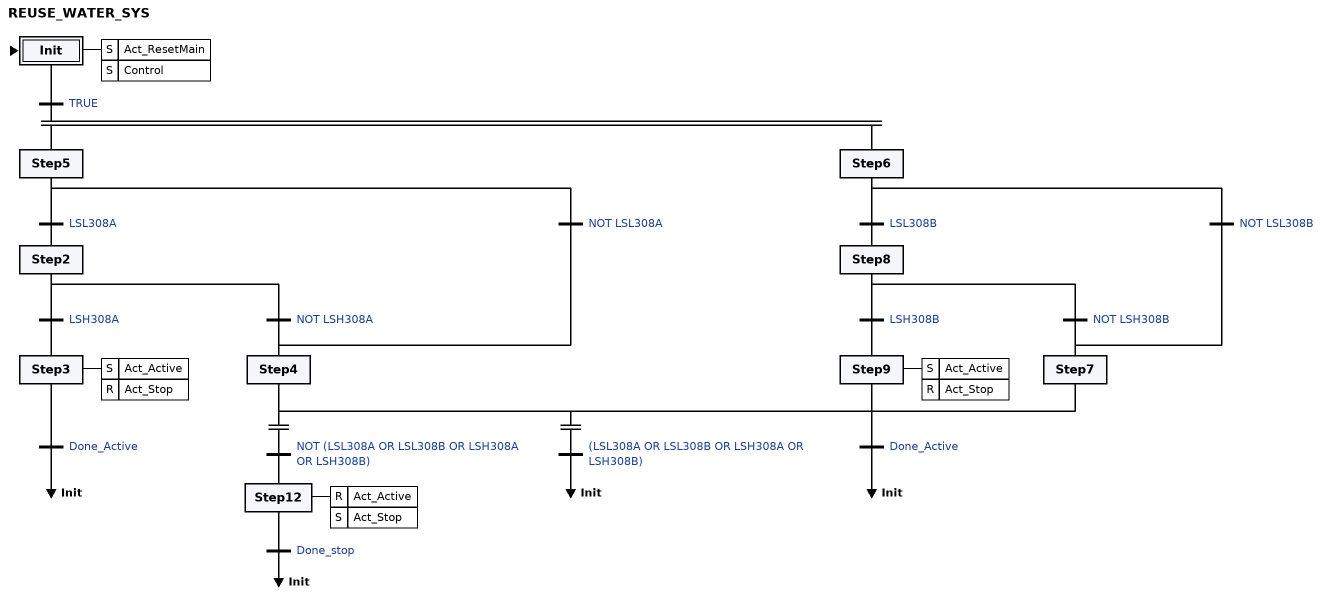
INITIAL_STEP Init:
	Act_ResetMain(S);
	Control(S);
END_STEP
TRANSITION FROM Init TO (Step5, Step6) := TRUE;
END_TRANSITION
STEP Step5:
END_STEP
TRANSITION FROM Step5 TO Step2 := LSL308A;
END_TRANSITION
TRANSITION FROM Step5 TO Step4 := NOT LSL308A;
END_TRANSITION
STEP Step2:
END_STEP
TRANSITION FROM Step2 TO Step3 := LSH308A;
END_TRANSITION
TRANSITION FROM Step2 TO Step4 := NOT LSH308A;
END_TRANSITION
STEP Step3:
	Act_Active(S);
	Act_Stop(R);
END_STEP
TRANSITION FROM Step3 TO Init := Done_Active;
END_TRANSITION
STEP Step4:
END_STEP
STEP Step6:
END_STEP
TRANSITION FROM Step6 TO Step8 := LSL308B;
END_TRANSITION
TRANSITION FROM Step6 TO Step7 := NOT LSL308B;
END_TRANSITION
STEP Step8:
END_STEP
TRANSITION FROM Step8 TO Step9 := LSH308B;
END_TRANSITION
TRANSITION FROM Step8 TO Step7 := NOT LSH308B;
END_TRANSITION
STEP Step9:
	Act_Active(S);
	Act_Stop(R);
END_STEP
TRANSITION FROM Step9 TO Init := Done_Active;
END_TRANSITION
STEP Step7:
END_STEP
TRANSITION FROM (Step4, Step7) TO Step12 := NOT (LSL308A OR LSL308B OR LSH308A OR LSH308B);
END_TRANSITION
TRANSITION FROM (Step4, Step7) TO Init := (LSL308A OR LSL308B OR LSH308A OR LSH308B);
END_TRANSITION
STEP Step12:
	Act_Active(R);
	Act_Stop(S);
END_STEP
TRANSITION FROM Step12 TO Init := Done_stop;
END_TRANSITION
END_FUNCTION_BLOCK
ACTION Act_Active:
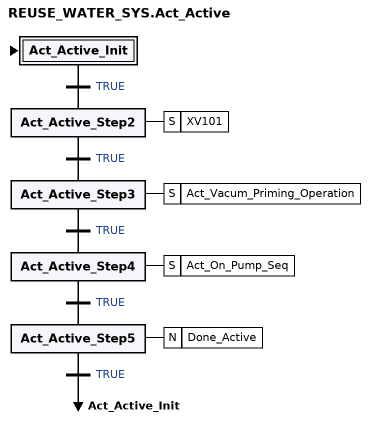
INITIAL_STEP Act_Active_Init:
END_STEP
TRANSITION FROM Act_Active_Init TO Act_Active_Step2 := TRUE;
END_TRANSITION
STEP Act_Active_Step2:
	XV101(S);
END_STEP
TRANSITION FROM Act_Active_Step2 TO Act_Active_Step3 := TRUE;
END_TRANSITION
STEP Act_Active_Step3:
	Act_Vacum_Priming_Operation(S);
END_STEP
TRANSITION FROM Act_Active_Step3 TO Act_Active_Step4 := TRUE;
END_TRANSITION
STEP Act_Active_Step4:
	Act_On_Pump_Seq(S);
END_STEP
TRANSITION FROM Act_Active_Step4 TO Act_Active_Step5 := TRUE;
END_TRANSITION
STEP Act_Active_Step5:
	Done_Active(N);
END_STEP
TRANSITION FROM Act_Active_Step5 TO Act_Active_Init := TRUE;
END_TRANSITION
END_ACTION
ACTION Act_On_Pump_Seq:
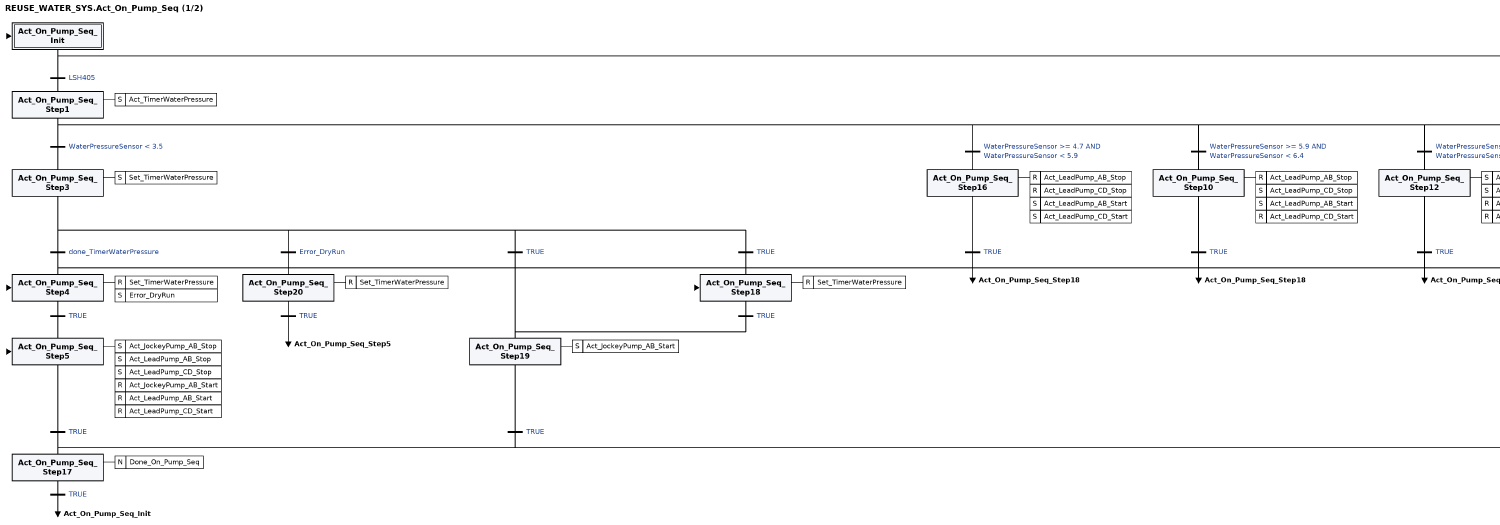
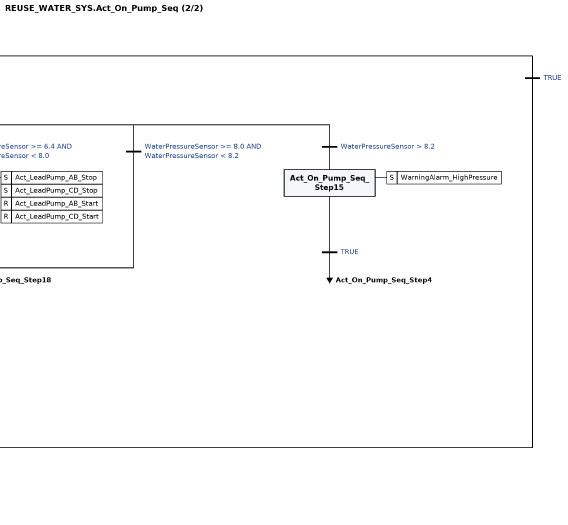
INITIAL_STEP Act_On_Pump_Seq_Init:
END_STEP
TRANSITION FROM Act_On_Pump_Seq_Init TO Act_On_Pump_Seq_Step1 := LSH405;
END_TRANSITION
TRANSITION FROM Act_On_Pump_Seq_Init TO Act_On_Pump_Seq_Step17 := TRUE;
END_TRANSITION
STEP Act_On_Pump_Seq_Step1:
	Act_TimerWaterPressure(S);
END_STEP
TRANSITION FROM Act_On_Pump_Seq_Step1 TO Act_On_Pump_Seq_Step3 := WaterPressureSensor < 3.5;
END_TRANSITION
TRANSITION FROM Act_On_Pump_Seq_Step1 TO Act_On_Pump_Seq_Step16 := WaterPressureSensor >= 4.7 AND WaterPressureSensor < 5.9;
END_TRANSITION
TRANSITION FROM Act_On_Pump_Seq_Step1 TO Act_On_Pump_Seq_Step10 := WaterPressureSensor >= 5.9 AND WaterPressureSensor < 6.4;
END_TRANSITION
TRANSITION FROM Act_On_Pump_Seq_Step1 TO Act_On_Pump_Seq_Step12 := WaterPressureSensor >= 6.4 AND WaterPressureSensor < 8.0;
END_TRANSITION
TRANSITION FROM Act_On_Pump_Seq_Step1 TO Act_On_Pump_Seq_Step4 := WaterPressureSensor >= 8.0 AND WaterPressureSensor < 8.2;
END_TRANSITION
TRANSITION FROM Act_On_Pump_Seq_Step1 TO Act_On_Pump_Seq_Step15 := WaterPressureSensor > 8.2;
END_TRANSITION
STEP Act_On_Pump_Seq_Step3:
	Set_TimerWaterPressure(S);
END_STEP
TRANSITION FROM Act_On_Pump_Seq_Step3 TO Act_On_Pump_Seq_Step4 := done_TimerWaterPressure;
END_TRANSITION
TRANSITION FROM Act_On_Pump_Seq_Step3 TO Act_On_Pump_Seq_Step20 := Error_DryRun;
END_TRANSITION
TRANSITION FROM Act_On_Pump_Seq_Step3 TO Act_On_Pump_Seq_Step19 := TRUE;
END_TRANSITION
TRANSITION FROM Act_On_Pump_Seq_Step3 TO Act_On_Pump_Seq_Step18 := TRUE;
END_TRANSITION
STEP Act_On_Pump_Seq_Step4:
	Set_TimerWaterPressure(R);
	Error_DryRun(S);
END_STEP
TRANSITION FROM Act_On_Pump_Seq_Step4 TO Act_On_Pump_Seq_Step5 := TRUE;
END_TRANSITION
STEP Act_On_Pump_Seq_Step5:
	Act_JockeyPump_AB_Stop(S);
	Act_LeadPump_AB_Stop(S);
	Act_LeadPump_CD_Stop(S);
	Act_JockeyPump_AB_Start(R);
	Act_LeadPump_AB_Start(R);
	Act_LeadPump_CD_Start(R);
END_STEP
TRANSITION FROM Act_On_Pump_Seq_Step5 TO Act_On_Pump_Seq_Step17 := TRUE;
END_TRANSITION
STEP Act_On_Pump_Seq_Step20:
	Set_TimerWaterPressure(R);
END_STEP
TRANSITION FROM Act_On_Pump_Seq_Step20 TO Act_On_Pump_Seq_Step5 := TRUE;
END_TRANSITION
STEP Act_On_Pump_Seq_Step18:
	Set_TimerWaterPressure(R);
END_STEP
TRANSITION FROM Act_On_Pump_Seq_Step18 TO Act_On_Pump_Seq_Step19 := TRUE;
END_TRANSITION
STEP Act_On_Pump_Seq_Step19:
	Act_JockeyPump_AB_Start(S);
END_STEP
TRANSITION FROM Act_On_Pump_Seq_Step19 TO Act_On_Pump_Seq_Step17 := TRUE;
END_TRANSITION
STEP Act_On_Pump_Seq_Step16:
	Act_LeadPump_AB_Stop(R);
	Act_LeadPump_CD_Stop(R);
	Act_LeadPump_AB_Start(S);
	Act_LeadPump_CD_Start(S);
END_STEP
TRANSITION FROM Act_On_Pump_Seq_Step16 TO Act_On_Pump_Seq_Step18 := TRUE;
END_TRANSITION
STEP Act_On_Pump_Seq_Step10:
	Act_LeadPump_AB_Stop(R);
	Act_LeadPump_CD_Stop(S);
	Act_LeadPump_AB_Start(S);
	Act_LeadPump_CD_Start(R);
END_STEP
TRANSITION FROM Act_On_Pump_Seq_Step10 TO Act_On_Pump_Seq_Step18 := TRUE;
END_TRANSITION
STEP Act_On_Pump_Seq_Step12:
	Act_LeadPump_AB_Stop(S);
	Act_LeadPump_CD_Stop(S);
	Act_LeadPump_AB_Start(R);
	Act_LeadPump_CD_Start(R);
END_STEP
TRANSITION FROM Act_On_Pump_Seq_Step12 TO Act_On_Pump_Seq_Step18 := TRUE;
END_TRANSITION
STEP Act_On_Pump_Seq_Step15:
	WarningAlarm_HighPressure(S);
END_STEP
TRANSITION FROM Act_On_Pump_Seq_Step15 TO Act_On_Pump_Seq_Step4 := TRUE;
END_TRANSITION
STEP Act_On_Pump_Seq_Step17:
	Done_On_Pump_Seq(N);
END_STEP
TRANSITION FROM Act_On_Pump_Seq_Step17 TO Act_On_Pump_Seq_Init := TRUE;
END_TRANSITION
END_ACTION
ACTION Act_ResetMain:
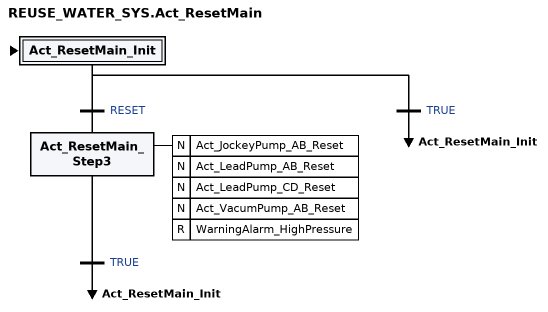
INITIAL_STEP Act_ResetMain_Init:
END_STEP
TRANSITION FROM Act_ResetMain_Init TO Act_ResetMain_Step3 := RESET;
END_TRANSITION
TRANSITION FROM Act_ResetMain_Init TO Act_ResetMain_Init := TRUE;
END_TRANSITION
STEP Act_ResetMain_Step3:
	Act_JockeyPump_AB_Reset(N);
	Act_LeadPump_AB_Reset(N);
	Act_LeadPump_CD_Reset(N);
	Act_VacumPump_AB_Reset(N);
	WarningAlarm_HighPressure(R);
END_STEP
TRANSITION FROM Act_ResetMain_Step3 TO Act_ResetMain_Init := TRUE;
END_TRANSITION
END_ACTION
ACTION Act_Stop:
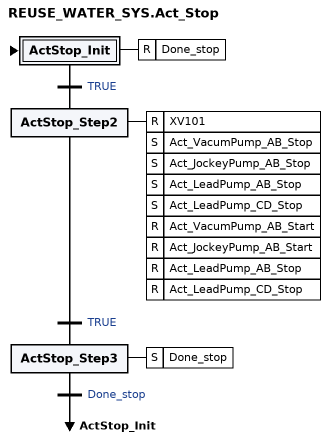
INITIAL_STEP ActStop_Init:
	Done_stop(R);
END_STEP
TRANSITION FROM ActStop_Init TO ActStop_Step2 := TRUE;
END_TRANSITION
STEP ActStop_Step2:
	XV101(R);
	Act_VacumPump_AB_Stop(S);
	Act_JockeyPump_AB_Stop(S);
	Act_LeadPump_AB_Stop(S);
	Act_LeadPump_CD_Stop(S);
	Act_VacumPump_AB_Start(R);
	Act_JockeyPump_AB_Start(R);
	Act_LeadPump_AB_Stop(R);
	Act_LeadPump_CD_Stop(R);
END_STEP
TRANSITION FROM ActStop_Step2 TO ActStop_Step3 := TRUE;
END_TRANSITION
STEP ActStop_Step3:
	Done_stop(S);
END_STEP
TRANSITION FROM ActStop_Step3 TO ActStop_Init := Done_stop;
END_TRANSITION
END_ACTION
ACTION Act_TimerWaterPressure:
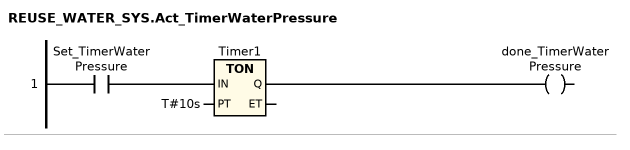
_LD_ (* Ladder Diagram *)
NETWORK 1
	[Set_TimerWaterPressure] - Timer1:TON(IN: *, PT: T#10s) --- (done_TimerWaterPressure)
_END_LD_
(* the same logic as Structured Text *)
(* Network 1 *)
Timer1(IN := Set_TimerWaterPressure, PT := T#10s);
done_TimerWaterPressure := Timer1.Q;
END_ACTION
ACTION Act_Vacum_Priming_Operation:
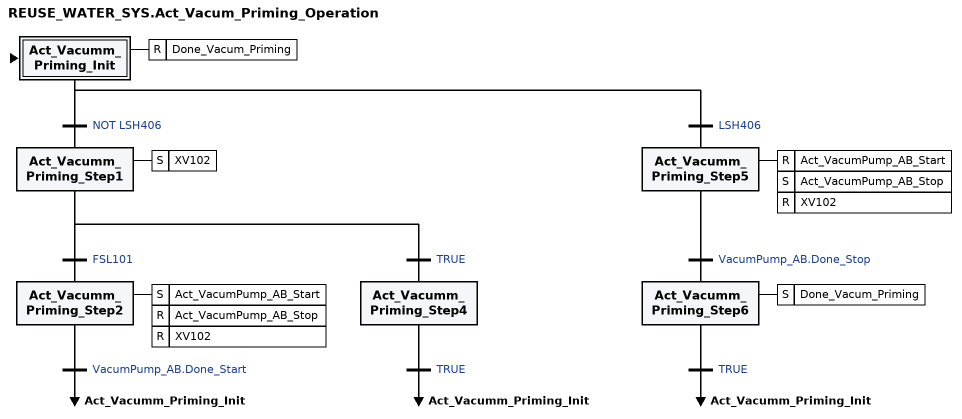
INITIAL_STEP Act_Vacumm_Priming_Init:
	Done_Vacum_Priming(R);
END_STEP
TRANSITION FROM Act_Vacumm_Priming_Init TO Act_Vacumm_Priming_Step1 := NOT LSH406;
END_TRANSITION
TRANSITION FROM Act_Vacumm_Priming_Init TO Act_Vacumm_Priming_Step5 := LSH406;
END_TRANSITION
STEP Act_Vacumm_Priming_Step1:
	XV102(S);
END_STEP
TRANSITION FROM Act_Vacumm_Priming_Step1 TO Act_Vacumm_Priming_Step2 := FSL101;
END_TRANSITION
TRANSITION FROM Act_Vacumm_Priming_Step1 TO Act_Vacumm_Priming_Step4 := TRUE;
END_TRANSITION
STEP Act_Vacumm_Priming_Step2:
	Act_VacumPump_AB_Start(S);
	Act_VacumPump_AB_Stop(R);
	XV102(R);
END_STEP
TRANSITION FROM Act_Vacumm_Priming_Step2 TO Act_Vacumm_Priming_Init := VacumPump_AB.Done_Start;
END_TRANSITION
STEP Act_Vacumm_Priming_Step4:
END_STEP
TRANSITION FROM Act_Vacumm_Priming_Step4 TO Act_Vacumm_Priming_Init := TRUE;
END_TRANSITION
STEP Act_Vacumm_Priming_Step5:
	Act_VacumPump_AB_Start(R);
	Act_VacumPump_AB_Stop(S);
	XV102(R);
END_STEP
TRANSITION FROM Act_Vacumm_Priming_Step5 TO Act_Vacumm_Priming_Step6 := VacumPump_AB.Done_Stop;
END_TRANSITION
STEP Act_Vacumm_Priming_Step6:
	Done_Vacum_Priming(S);
END_STEP
TRANSITION FROM Act_Vacumm_Priming_Step6 TO Act_Vacumm_Priming_Init := TRUE;
END_TRANSITION
END_ACTION
ACTION Act_VacumPump_AB_Reset:
